// TwinCAT 3 PLC project PLC
// Title: ADO_Demo_PLC
// Company: Beckhoff
// ProjectVersion: 0.0.1
// ProgramVersion: 3.1.4024.0
// libraries:
//   Tc2_Standard, * (Beckhoff Automation GmbH)
//   Tc2_System, * (Beckhoff Automation GmbH)
//   Tc3_Module, * (Beckhoff Automation GmbH)
// project tree:
//   DUTs/ E_AutoMan.TcDUT (not stored), ST_CellConfig.TcDUT (not stored), ST_PartStatus.TcDUT (not stored)
//   / GlobalTextList.TcGTLO (not stored), PlcTask.TcTTO
//   POUs/Cell/ E_CellState.TcDUT (not stored), FB_Cell.TcPOU
//   POUs/Devices/ FB_Axis.TcPOU (not stored), FB_Actuator.TcPOU (not stored), IActuator.TcIO (not stored), IAxis.TcIO (not stored)
//   POUs/ MAIN.TcPOU (not stored)
//   POUs/Stations/ E_StationState.TcDUT (not stored), FB_BarcodeScanner.TcPOU (not stored), FB_Filler.TcPOU (not stored), FB_Capper.TcPOU (not stored), FB_CheckWeigher.TcPOU (not stored), FB_Station.TcPOU (not stored), IStation.TcIO (not stored)
//   TestFramework/ FB_Test.TcPOU, ITest.TcIO, ST_TestResults.TcDUT
//   Tests/ FB_TEST_CheckPartGood.TcPOU, FB_TEST_CheckPartCapperFail.TcPOU, FB_TEST_CheckPartBarcodeFail.TcPOU, FB_TEST_CheckPartFillerFail.TcPOU, PRG_TEST.TcPOU
// real-time tasks:
//   TASK PlcTask: cycle T#10ms, priority 20, ADS port 350

CONFIGURATION PLC
    RESOURCE PLC ON TwinCAT3
        TASK PlcTask(INTERVAL := T#10ms, PRIORITY := 20);
        PROGRAM PRG_TEST WITH PlcTask : PRG_TEST;
    END_RESOURCE
END_CONFIGURATION

// ---- TestFramework/ST_TestResults.TcDUT
TYPE ST_TestResults :
STRUCT
	Result		: BOOL;
	Message		: STRING(255);
END_STRUCT
END_TYPE

// ---- TestFramework/ITest.TcIO
INTERFACE ITest

METHOD Execute : ST_TestResults
VAR_INPUT
END_VAR
END_METHOD

END_INTERFACE

// ---- Tests/PRG_TEST.TcPOU
PROGRAM PRG_TEST
VAR
	fbCheckPartGood				: FB_TEST_CheckPartGood;
	fbCheckPartCapperFail		: FB_TEST_CheckPartCapperFail;
	fbCheckPartBarcodeFail		: FB_TEST_CheckPartBarcodeFail;
	fbCheckPartFillerFail		: FB_TEST_CheckPartFillerFail;
END_VAR

END_PROGRAM

// ---- Tests/FB_TEST_CheckPartGood.TcPOU
FUNCTION_BLOCK FB_TEST_CheckPartGood EXTENDS FB_Test
VAR
END_VAR

METHOD Execute : ST_TestResults
VAR
	MockStatus		: ST_PartStatus;
	fbCell			: FB_Cell;
	testExpected	: BOOL;
	testResult		: BOOL;
END_VAR
MockStatus.bBarcodeStatus := TRUE;
MockStatus.bCapperStatus := TRUE;
MockStatus.bFillerStatus := TRUE;
MockStatus.bWeightStatus := TRUE;

testExpected := TRUE;
testResult := fbCell.CheckPart(MockStatus);

Execute := AssertEquals(
	testExpected, 
	testResult, 
	'CheckPart Part status expected true, returned false.'
);
END_METHOD

END_FUNCTION_BLOCK

// ---- TestFramework/FB_Test.TcPOU
FUNCTION_BLOCK ABSTRACT FB_Test IMPLEMENTS ITest
VAR
END_VAR

METHOD PROTECTED AssertEquals : ST_TestResults
VAR_INPUT
	expected		: ANY;
	result			: ANY;
	failmsg			: STRING(255);
END_VAR
VAR
	sExp, sRes		: STRING;
	results			: ST_TestResults;
END_VAR
IF (expected.diSize <> result.diSize) THEN
	results.Message := 'Test error: expected value type mismatch';
	results.Result := FALSE;
	AssertEquals := results;
	RETURN;
END_IF

IF (Expected.pValue^ <> Result.pValue^) THEN
	sExp := CONCAT(' Expected: ', TO_STRING(expected.pValue^));
	sRes := CONCAT(' Result: ', TO_STRING(result.pValue^));
	results.Message := CONCAT(CONCAT(failmsg, sExp), sRes);
	results.Result := FALSE;
	AssertEquals := results;
ELSE
	results.Result := TRUE;
	AssertEquals := results;
END_IF
END_METHOD

{attribute 'TcRpcEnable'}
METHOD Execute : ST_TestResults;
VAR
END_VAR
END_METHOD

END_FUNCTION_BLOCK

// ---- POUs/Cell/FB_Cell.TcPOU
FUNCTION_BLOCK FB_Cell
VAR_INPUT
END_VAR
VAR_OUTPUT
END_VAR
VAR
	eAutoMan					: E_AutoMan := E_AutoMan.AUTO;
	State						: E_CellState;
	
	// IO
	bStartBtn					AT %I* : BOOL;
	bStopBtn					AT %I* : BOOL;
	bPartPresentAtInfeed		AT %I* : BOOL;
	bPartPresentAtOutfeed		AT %I* : BOOL;
	
	{attribute 'TcAnalytics'}
	fFillRate					AT %Q* : LREAL := 2.5;
	
	// devices
	fbInfeedActuator			: FB_Actuator;
	fbOutfeedActuator			: FB_Actuator;
	fbInfeedConveyor			: FB_Axis;
	fbIndexConveyor				: FB_Axis;
	fbOutfeedConveyor			: FB_Axis;
	
	InfeedConveyor				: IAxis := fbInfeedConveyor;
	IndexConveyor				: IAxis := fbIndexConveyor;
	InfeedActuator				: IActuator := fbInfeedActuator;
	OutfeedActuator				: IActuator := fbOutfeedActuator;
	OutfeedConveyor				: IAxis := fbOutfeedConveyor;
	
	// stations
	fbBarcoder					: FB_BarcodeScanner;
	fbFiller					: FB_Filler;
	fbCapper					: FB_Capper;
	fbCheckWeigher				: FB_CheckWeigher;
	Stations					: ARRAY[0..3] OF IStation := [fbBarcoder, fbFiller, fbCapper, fbCheckWeigher];
	iStationCount				: DINT := 4;
	i							: DINT;
	
	bAllStationsReady			: BOOL;
	bCellPartPresent			: BOOL;
	bStationFaulted				: BOOL;
	tmrStationWait				: TON;
	bInFeeding					: BOOL;
	bIndexing					: BOOL;
	bOutfeeding					: BOOL;
	
	PartStatus					: ARRAY[0..3] OF ST_PartStatus;
	NewPart						: ST_PartStatus;
	
	{attribute 'TcAnalytics'}
	OutfeedPart					: ST_PartStatus;
	
	fIndexPosition				: LREAL;
	INDEX_DIST					: LREAL := 300.0;
	INDEX_VEL					: LREAL := 100.0;
	INFEED_VEL					: LREAL := 100.0;
	
	bStartReq					: BOOL;
	bStopReq					: BOOL;
	bInit 						: BOOL := TRUE;
	
	bFillRateTest				: BOOL;
	tmrFillRate					: TON;
END_VAR

METHOD PUBLIC CheckPart : BOOL
VAR_INPUT
	Status			: ST_PartStatus;
END_VAR
CheckPart := Status.bBarcodeStatus AND Status.bFillerStatus AND Status.bCapperStatus AND Status.bWeightStatus;
END_METHOD

METHOD PUBLIC Execute : PVOID
StationMgr();

IF eAutoMan = E_AutoMan.AUTO THEN
	
	CASE State OF
		
		E_CellState.STOPPED:
			
			IF bStartReq THEN
				State := E_CellState.IDLE_WAIT;
				bStartReq := FALSE;
			END_IF
			
		E_CellState.IDLE_WAIT:
		
			IF bPartPresentAtInfeed AND Stations[0] <> 0 
			AND (Stations[0].Ready AND NOT Stations[0].PartPresent) THEN
				State := E_CellState.FEED;
			END_IF
			
			IF bAllStationsReady AND bCellPartPresent THEN
				tmrStationWait(IN:=TRUE, PT:=T#500MS);
				IF tmrStationWait.Q THEN
					tmrStationWait(IN:=FALSE);
					State := E_CellState.INDEX;
				END_IF
			END_IF
			
			IF bStopReq THEN
				State := E_CellState.STOPPED;
				bStopReq := FALSE;
			END_IF
			
		E_CellState.FEED:
		
			IF NOT bInFeeding THEN
				MEMCPY(ADR(PartStatus[0]), ADR(NewPart), SIZEOF(ST_PartStatus));
				bInFeeding := TRUE;
			END_IF
			
			IF InfeedActuator.Cycle() THEN
				State := E_CellState.IDLE_WAIT;
				bInFeeding := FALSE;
			END_IF
			
		E_CellState.INDEX:
			
			IF NOT bIndexing THEN
				fIndexPosition := IndexConveyor.ActPosition + INDEX_DIST;
				bIndexing := TRUE;
			END_IF
			
			IF (IndexConveyor.MoveAbsolute(fIndexPosition, INDEX_VEL)) AND bIndexing THEN
				bIndexing := FALSE;
				OutfeedPart := PartStatus[3];
				MEMCPY(ADR(PartStatus[1]), ADR(PartStatus[0]), SIZEOF(ST_PartStatus)*3);
				MEMSET(ADR(PartStatus[0]), 0, SIZEOF(ST_PartStatus));
				State := E_CellState.IDLE_WAIT;
			END_IF
			
	END_CASE
	
	IF State <> E_CellState.STOPPED THEN
		
		InfeedConveyor.JogFwd(INFEED_VEL);
		OutfeedConveyor.JogFwd(INFEED_VEL);
		
		IF bPartPresentAtOutfeed THEN
			// bad part
			IF NOT CheckPart(OutfeedPart) THEN
				bOutFeeding := TRUE;
			END_IF
		END_IF
		IF bOutfeeding THEN
			IF OutfeedActuator.Cycle() THEN
				bOutfeeding := FALSE;
			END_IF
		END_IF
		
		IF bFillRateTest THEN
			tmrFillRate(IN:=NOT tmrFillRate.Q, PT:=T#20M); 
			IF tmrFillRate.Q THEN
				fFillRate := fFillRate + 0.05;
			END_IF
		END_IF
		
	ELSE
		InfeedConveyor.StopMove();
		OutfeedConveyor.StopMove();
	END_IF
	
END_IF

IF bStartBtn THEN
	bStopReq := FALSE;
	bStartReq := TRUE;
END_IF

IF bStopBtn THEN
	bStartReq := FALSE;
	bStopReq := TRUE;
END_IF
END_METHOD

METHOD PRIVATE StationMgr : PVOID
VAR_INPUT
END_VAR
IF iStationCount < 1 THEN
	RETURN;
END_IF

IF bInit THEN
	FOR i:= 0 TO iStationCount - 1 DO
		Stations[i].PartStatus := ADR(PartStatus[i]);
	END_FOR
	bInit := FALSE;
	bStartReq := TRUE;
END_IF

bAllStationsReady := TRUE;
bStationFaulted := FALSE;
bCellPartPresent := FALSE;

FOR i := 0 TO iStationCount - 1	DO
	IF (Stations[i] = 0) THEN
		CONTINUE;
	END_IF
	
	Stations[i].Execute();
	
	IF NOT Stations[i].Ready THEN
		bAllStationsReady := FALSE;
	END_IF
	
	IF Stations[i].Faulted THEN
		bStationFaulted := TRUE;
	END_IF
	
	IF Stations[i].PartPresent THEN
		bCellPartPresent := TRUE;
	END_IF
	
END_FOR
END_METHOD

END_FUNCTION_BLOCK

// ---- Tests/FB_TEST_CheckPartCapperFail.TcPOU
FUNCTION_BLOCK FB_TEST_CheckPartCapperFail EXTENDS FB_Test
VAR
END_VAR

METHOD Execute : ST_TestResults
VAR
	MockStatus		: ST_PartStatus;
	fbCell			: FB_Cell;
	testExpected	: BOOL;
	testResult		: BOOL;
END_VAR
MockStatus.bBarcodeStatus := TRUE;
MockStatus.bCapperStatus := FALSE;
MockStatus.bFillerStatus := TRUE;
MockStatus.bWeightStatus := TRUE;

testExpected := FALSE;
testResult := fbCell.CheckPart(MockStatus);

Execute := AssertEquals(
	testExpected, 
	testResult, 
	'Part status fail.'
);
END_METHOD

END_FUNCTION_BLOCK

// ---- Tests/FB_TEST_CheckPartBarcodeFail.TcPOU
FUNCTION_BLOCK FB_TEST_CheckPartBarcodeFail EXTENDS FB_Test
VAR
END_VAR

METHOD Execute : ST_TestResults
VAR
	MockStatus		: ST_PartStatus;
	fbCell			: FB_Cell;
	testExpected	: BOOL;
	testResult		: BOOL;
END_VAR
MockStatus.bBarcodeStatus := FALSE;
MockStatus.bCapperStatus := TRUE;
MockStatus.bFillerStatus := TRUE;
MockStatus.bWeightStatus := TRUE;

testExpected := FALSE;
testResult := fbCell.CheckPart(MockStatus);

Execute := AssertEquals(
	testExpected, 
	testResult, 
	'Part status fail.'
);
END_METHOD

END_FUNCTION_BLOCK

// ---- Tests/FB_TEST_CheckPartFillerFail.TcPOU
FUNCTION_BLOCK FB_TEST_CheckPartFillerFail EXTENDS FB_Test
VAR
END_VAR

METHOD Execute : ST_TestResults
VAR
	MockStatus		: ST_PartStatus;
	fbCell			: FB_Cell;
	testExpected	: BOOL;
	testResult		: BOOL;
END_VAR
MockStatus.bBarcodeStatus := TRUE;
MockStatus.bCapperStatus := TRUE;
MockStatus.bFillerStatus := TRUE;
MockStatus.bWeightStatus := TRUE;

testExpected := FALSE;
testResult := fbCell.CheckPart(MockStatus);

Execute := AssertEquals(
	testExpected, 
	testResult, 
	'Part status fail.'
);
END_METHOD

END_FUNCTION_BLOCK
